FUNCTION_BLOCK T_CylinderComponent EXTENDS FB_ComponentBase
VAR
	_cylinder : I_Cylinder;
END_VAR

METHOD GenericInitialise
VAR_INPUT
	Cylinder : I_Cylinder; 
END_VAR
_cylinder := Cylinder;
END_METHOD

END_FUNCTION_BLOCK

(* stored: Version 1.1.0.1, ProductVersion 3.1.4024.12
   POU T_CylinderComponent: Id {9c58672d-2584-427d-923c-5ff0608b9288}, SpecialFunc None
   Method GenericInitialise: Id {be4c08c4-f43f-4504-99bd-20dd1643bb74} *)
